(* IEC 61131-3 sources: canworks/test/fixtures/editor-project/pous/programs, 1 file *)

(* ---- main.st ---- *)
PROGRAM main
  VAR
    door_ok AT %IX10.1 : BOOL;
    counter : INT;
  END_VAR

  IF door_ok THEN
    counter := counter + 1;
  END_IF;
END_PROGRAM
